// TwinCAT 3 PLC project UDP
// ProgramVersion: 3.1.4022.0
// libraries:
//   Tc2_Standard, * (Beckhoff Automation GmbH)
//   Tc2_System, * (Beckhoff Automation GmbH)
//   Tc3_Module, * (Beckhoff Automation GmbH)
// project tree:
//   GVLs/ UDP.TcGVL
//   / PlcTask.TcTTO
//   POUs/ MAIN.TcPOU, UDPConnect.TcPOU
// (motion and I/O tree: see PLC project shutdown)
// real-time tasks:
//   TASK PlcTask: cycle T#10ms, priority 20, ADS port 350
//   TASK updateIrSensors: cycle T#5ms, priority 9, ADS port 351
//   TASK UDP Task: cycle T#10ms, priority 10, ADS port 354
// variable links:

CONFIGURATION UDP
    RESOURCE PLC ON TwinCAT3
        TASK PlcTask(INTERVAL := T#5ms, PRIORITY := 2);
        PROGRAM MAIN WITH PlcTask : MAIN;
    END_RESOURCE
END_CONFIGURATION

// ---- GVLs/UDP.TcGVL
{attribute 'qualified_only'}
VAR_GLOBAL
	sPaketinhalt	: LREAL;
	nPaketlaenge	: UDINT;
	
	x		: ARRAY[1..4] OF LREAL;
	y		: ARRAY[1..4] OF LREAL;
	theta	: ARRAY[1..4] OF LREAL;
END_VAR

// ---- POUs/MAIN.TcPOU
PROGRAM MAIN
VAR
	udp1 : UDPConnect;
END_VAR

udp1();

END_PROGRAM

// ---- POUs/UDPConnect.TcPOU
{attribute 'c++_compatible'}
FUNCTION_BLOCK UDPConnect IMPLEMENTS ITcIoUdpProtocolRecv
VAR_INPUT
END_VAR
VAR_OUTPUT
END_VAR
VAR
	{attribute 'TcInitSymbol'}
    oid:              OTCID; 
    ipUdp:            ITcIoUdpProtocol;
    updPort:          UINT := 25000;
    nReceivedPakets:  UINT;
    hrInit :          HRESULT;
    hrSend :          HRESULT;
END_VAR

IF ipUdp <> 0 THEN
    ipUdp.CheckReceived();
END_IF

METHOD FB_exit : BOOL
VAR_INPUT
	bInCopyCode : BOOL; // if TRUE, the exit method is called for exiting an instance that is copied afterwards (online change).
END_VAR
IF (NOT bInCopyCode AND ipUdp <> 0) THEN //Shutdown
     ipUdp.UnregisterReceiver(updPort);
    FW_SafeRelease(ADR(ipUdp));
     FB_exit := TRUE;
ELSE
     FB_exit := FALSE;
END_IF
END_METHOD

METHOD FB_init : BOOL
VAR_INPUT
	bInitRetains : BOOL; // if TRUE, the retain variables are initialized (warm start / cold start)
	bInCopyCode : BOOL;  // if TRUE, the instance afterwards gets moved into the copy code (online change)
END_VAR

VAR
    ipSrv: ITComObjectServer;
    hr : HRESULT;
END_VAR
IF NOT bInCopyCode THEN // no online change
    IF ipUdp = 0 THEN
     hrInit := FW_ObjMgr_GetObjectInstance(   oid:=oid, 
    
    iid:=TC_GLOBAL_IID_LIST.IID_ITcIoUdpProtocol, 

    pipUnk:=ADR(ipUdp) );
        IF ( SUCCEEDED(hr) AND ipUdp.RegisterReceiver(updPort, THIS^) = 0 ) THEN //open port
            FB_init := TRUE;
        ELSE
            FB_init := FALSE; 
            FW_SafeRelease(ADR(ipUdp));
        END_IF
    END_IF
END_IF
END_METHOD

METHOD FB_reinit : BOOL
VAR_INPUT
END_VAR
IF (ipUdp <> 0) THEN 
 ipUdp.RegisterReceiver(updPort, THIS^);
END_IF
END_METHOD

{attribute 'object_name' := 'ReceiveData'}
{attribute 'c++_compatible'}
{attribute 'signature_flag' := '33554688'}
{attribute 'pack_mode' := '4'}
{attribute 'show'}
{attribute 'minimal_input_size' := '4'}
METHOD ReceiveData : HRESULT
VAR_INPUT
	ipAddr	: UDINT;
	udpDestPort	: UINT;
	udpSrcPort	: UINT;
	nData	: UDINT;
	pData	: PVOID;
	pVlan	: POINTER TO ETYPE_VLAN_HEADER := 0;
END_VAR

VAR
	nEmpfangen		: UINT;

	UDPVariablen: INT;
END_VAR
nReceivedPakets := nReceivedPakets+1;
UDP.nPaketlaenge := nData;

memcpy(ADR(UDP.x[1]),pData,8);
memcpy(ADR(UDP.y[1]),pData+8,8);
memcpy(ADR(UDP.theta[1]),pData+16,8);
END_METHOD

{attribute 'c++_compatible'}
{attribute 'minimal_input_size' := '4'}
{attribute 'pack_mode' := '4'}
{warning 'Methodenimplementierung hinzufügen'}
METHOD TcAddRef : UDINT
END_METHOD

{attribute 'c++_compatible'}
{attribute 'minimal_input_size' := '4'}
{attribute 'pack_mode' := '4'}
{warning 'Methodenimplementierung hinzufügen'}
METHOD TcQueryInterface : HRESULT
VAR_INPUT
	iid	: REFERENCE TO IID;
	pipItf	: POINTER TO PVOID;
END_VAR
END_METHOD

{attribute 'c++_compatible'}
{attribute 'minimal_input_size' := '4'}
{attribute 'pack_mode' := '4'}
{warning 'Methodenimplementierung hinzufügen'}
METHOD TcRelease : UDINT
END_METHOD

END_FUNCTION_BLOCK
